// TIA Portal V15.1 export
// export: Created 2024-06-21T08:41:11.6388979Z, ExportSetting WithDefaults, DisplayName Totally Integrated Automation Portal, DisplayVersion V15.1 Update 5, DisplayName TIA Portal Openness, DisplayVersion V15.1 Update 5, DisplayName SINAMICS Startdrive Advanced, DisplayVersion V15.1, DisplayName G130, G150, S120, S150, SINAMICS MV, S210, DisplayVersion V15.1, DisplayName G110M, G120, G120C, G120D, G120P, DisplayVersion V15.1, DisplayName STEP 7 Professional, DisplayVersion V15.1 Update 5, DisplayName STEP 7 Safety, DisplayVersion V15.1, DisplayName WinCC Professional, DisplayVersion V15.1 Update 5, DisplayName SIMATIC Visualization Architect, DisplayVersion V15.1
FUNCTION "LGBValveStatus" : Void   // FC6620, SCL
{ S7_Optimized_Access := 'TRUE' }
VERSION : 0.1
// stored: AutoNumber false, IsIECCheckEnabled false, SetENOAutomatically False, UDAEnableTagReadback false
   VAR_IN_OUT
      IO_Pipe : Array[1..50] of "TCPipe";
      IO_Valve : Array[1..50] of "TCValve";
   END_VAR
   VAR_TEMP
      RetVal : Int;
      Pipe : Int;
   END_VAR
BEGIN

   FOR #Pipe := 1 TO 50 DO
       "LGBValveStatusSub"(PipeData := #IO_Pipe[#Pipe]  // IN: UDT
                           , ValveStatus => #IO_Valve[#Pipe]  // OUT: UDT
       ); // VOID  
   END_FOR;
END_FUNCTION
